PROGRAM LIGHTLOGIC
VAR
	
	REDSTACK	:BLINK;
	AMBERSTACK	:BLINK;
	
	LIGHTS		:INT;

END_VAR

(*RESET LED*)
(*RESET LED ON IF ATTACHMENT GOES INTO E-STOP STATE*)

IF MOBILEHOIST.ESTOP_CONDITION THEN
	
	MOBILEHOIST.RESETPB_LED 	:= TRUE;

ELSE

	MOBILEHOIST.RESETPB_LED		:= FALSE;

END_IF

(*RED STACK LIGHT LED*)
(*RED STACK LIGHT LED ON IF ATTACHMENT GOES INTO E-STOP STATE*)
IF MOBILEHOIST.ESTOP_CONDITION THEN
	
	MOBILEHOIST.REDSTACKLIGHT 	:= TRUE;

(*RED STACK LIGHT LED BLINK IF ATTACHMENT LOSE CONNECTIVITY BETWEEN IO CARDS*)
ELSIF MOBILEHOIST.IOERROR THEN
	

	REDSTACK(ENABLE:= TRUE , PERIOD:= T#500MS , Q=> MOBILEHOIST.REDSTACKLIGHT);

ELSE
	
	MOBILEHOIST.REDSTACKLIGHT 	:=FALSE;
	
END_IF

(*AMBER STACK LIGHT LED*)
(*AMBER STACK LIGHT LED ON IF IMPROPERLY LOWERED IN THE GROUND*)
IF MOBILEHOIST.ESTOP_CONDITION = FALSE THEN

IF MOBILEHOIST.LOWERED_IMPROPERLY THEN
	
	MOBILEHOIST.AMBERSTACKLIGHT 	:=TRUE;

ELSE 

	MOBILEHOIST.AMBERSTACKLIGHT	:=FALSE;
	
END_IF

ELSIF MOBILEHOIST.ESTOP_CONDITION THEN
	
	MOBILEHOIST.AMBERSTACKLIGHT := FALSE;	

END_IF

(*GREEN LIGHT*)
(*GREEN SELECTOR SWITCH LIGHT ON IF ATTACHMENT IS OUT OF FAULTS*)
IF MOBILEHOIST.ESTOP_CONDITION = FALSE THEN
	
IF MOBILEHOIST.LOWERED_PROPERLY THEN
	
	MOBILEHOIST.SELECTORSW_LED := TRUE;
	
ELSE
	
	MOBILEHOIST.SELECTORSW_LED := FALSE;
	
END_IF

ELSIF MOBILEHOIST.ESTOP_CONDITION THEN
	
	MOBILEHOIST.SELECTORSW_LED := FALSE;
	
END_IF

(*DEADMAN LIGHT LED*)

IF MOBILEHOIST.ESTOP_CONDITION OR MOBILEHOIST.IOERROR	THEN
	
	MOBILEHOIST.REDSTACKLIGHT 	:= TRUE;

ELSIF MOBILEHOIST.DEADMAN_SWITCH THEN
	

	REDSTACK(ENABLE:= TRUE , PERIOD:= T#500MS , Q=> MOBILEHOIST.REDSTACKLIGHT);
	
	AMBERSTACK(ENABLE:= TRUE , PERIOD:= T#500MS , Q=> MOBILEHOIST.AMBERSTACKLIGHT);
	
END_IF

END_PROGRAM

(* stored: Version 1.1.0.1, ProductVersion 3.1.4024.11
   POU LIGHTLOGIC: Id {2d97790c-4942-4292-8cbe-2f4ff2397944}, SpecialFunc None *)
